TYPE DSV3_TempCtrlRecipe :
STRUCT
	Station: ARRAY [0..iStnQty] OF DSV3_TempCtrlParameter;

END_STRUCT
END_TYPE

(* stored: Version 1.1.0.1, ProductVersion 3.1.4024.12
   DUT DSV3_TempCtrlRecipe: Id {96dfa11f-4dc0-497c-b0c9-58ac52114b02} *)
